FUNCTION_BLOCK FB_GripAngleCalc
VAR_INPUT
END_VAR
VAR_OUTPUT
END_VAR
VAR
	// limit value
	m_minHallSensorValue :LREAL;
	m_maxHallSensorValue:LREAL;
	m_hallSensorRange:LREAL;
	
	// grip angle from hall sensor IO
	m_gripHallSenorValue :LREAL;
	m_normHallSensorValue: LREAL;
	m_gripAngle :LREAL;
	m_gripAngLpf : FB_LowPassFilter;
END_VAR

METHOD init : BOOL
VAR_INPUT
	i_armIdx:INT;
END_VAR
// init limit value
m_minHallSensorValue:=(GVL_ArmJointCaliData.g_minHallSensorValue[i_armIdx]/65536) AND 16#0000FFFF; 
m_maxHallSensorValue:=(GVL_ArmJointCaliData.g_maxHallSensorValue[i_armIdx]/65536) AND 16#0000FFFF; 
m_hallSensorRange := m_maxHallSensorValue-m_minHallSensorValue;

// init filter
m_gripAngLpf.init(1, g_gripAngLpfCutoffFreq, g_armCtrlFreq);
END_METHOD

METHOD run : LREAL
VAR_INPUT
	IOValue : UDINT;
END_VAR
// sensor io parse
m_gripHallSenorValue:=(IOValue/65536) AND 16#0000FFFF; //high 16 bits

// normalize hall sensor value
m_normHallSensorValue:=LIMIT(0, (m_gripHallSenorValue-m_minHallSensorValue)/m_hallSensorRange, 1);

IF m_normHallSensorValue<=0.019 THEN
	// grip angle fitting
	m_gripAngle := g_masterGripAngleFitCoeff2[1] * EXPT(m_normHallSensorValue,3)
				+ g_masterGripAngleFitCoeff2[2] * EXPT(m_normHallSensorValue,2)
				+ g_masterGripAngleFitCoeff2[3] * EXPT(m_normHallSensorValue,1)
				+ g_masterGripAngleFitCoeff2[4];
ELSE
	m_gripAngle := g_masterGripAngleFitCoeff[1] * EXPT(m_normHallSensorValue,5)
			+ g_masterGripAngleFitCoeff[2] * EXPT(m_normHallSensorValue,4)
			+ g_masterGripAngleFitCoeff[3] * EXPT(m_normHallSensorValue,3)
			+ g_masterGripAngleFitCoeff[4] * EXPT(m_normHallSensorValue,2)
			+ g_masterGripAngleFitCoeff[5] * EXPT(m_normHallSensorValue,1)
			+ g_masterGripAngleFitCoeff[6];
END_IF


// filt and cap the result
m_gripAngle := m_gripAngLpf.run(m_gripAngle);
m_gripAngle := LIMIT(g_minGripAngle, m_gripAngle, g_maxGripAngle);

run:=m_gripAngle;
END_METHOD

END_FUNCTION_BLOCK

(* stored: Version 1.1.0.1, ProductVersion 3.1.4024.11
   POU FB_GripAngleCalc: Id {1d1f59c4-2943-4ee4-8e94-d36cfa692bb0}, SpecialFunc None
   Method init: Id {e4f56e13-70f8-4942-94ed-464230d0ebf2}
   Method run: Id {55aa24f7-dd28-41ed-8903-b3831602df36} *)
